TYPE AxesPointingModelsSetupStatuses :
STRUCT
	///Is the pointing models setup in a busy state?
	busyStatus: BusyStatus;
	///Is the pointing models setup in a healthy state?
	healthStatus: HealthStatus;
END_STRUCT
END_TYPE

(* stored: Version 1.1.0.1, ProductVersion 3.1.4019.2
   DUT AxesPointingModelsSetupStatuses: Id {f378df93-f5d5-405c-a9ad-64cf16cf49c7} *)
